// TIA Portal V17 export
// export: Created 2022-07-20T06:59:51.5033587Z, ExportSetting WithDefaults, DisplayName Totally Integrated Automation Portal, DisplayVersion V17, DisplayName TIA Portal Openness, DisplayVersion V17, DisplayName TIA Portal Version Control Interface, DisplayVersion V17, DisplayName SINAMICS Startdrive Advanced, DisplayVersion V17, DisplayName SINAMICS Startdrive G130, G150, S120, S150, SINAMICS MV, S210, DisplayVersion V17, DisplayName SINAMICS Startdrive G110M, G120, G120C, G120D, G120P, G115D, DisplayVersion V17, DisplayName STEP 7 Professional, DisplayVersion V17, DisplayName STEP 7 Safety, DisplayVersion V17, DisplayName WinCC Advanced, DisplayVersion V17
FUNCTION_BLOCK "FB10064_IperCleaningTrays"   // FB10064, LAD
{ S7_Optimized_Access := 'TRUE' }
VERSION : 0.1
// stored: AutoNumber false, IsIECCheckEnabled false, IsRetainMemResEnabled false, MemoryReserve 100, SetENOAutomatically false, UDAEnableTagReadback false
   VAR_INPUT
      Acknowledge : Bool;
      DriveInLexium : "TLexium_MDrv_Drv2Plc";
      RequestAcknowledge : Bool;
      CleaningTray_HomingSensor : Bool;
      CleaningTray_PurgeTrayPositionSensor_1 : Bool;
      CleaningTray_PurgeTrayPositionSensor_2 : Bool;
      PurgeTray1_HomingPositionSensor : Bool;
      PurgeTray2_HomingPositionSensor : Bool;
      PurgeTray1_PurgePositionSensor : Bool;
      PurgeTray2_PurgePositionSensor : Bool;
      Motor_HoldCurrent : SInt;
      Motor_RunCurrent : SInt;
      Motor_MmByMotorTurn : Real;
      Motor_HomingSpeedMmBySec : Real;
      Motor_SpeedMmBySec : Real;
      Motor_AccelerationMmBySec2 : DInt;
      Motor_DecelerationMmBySec2 : DInt;
      Motor_JogSpeedMmBySec : Real;
      Motor_RequestStop : Bool;
      CleaningTray_HomingPosition : Real;
      CleaningTray_CleaningPosition_1 : Real;
      CleaningTray_CleaningPosition_2 : Real;
      CleaningTray_WipingPosition_1 : Real;
      CleaningTray_WipingPosition_2 : Real;
      CleaningTray_RequestHoming : Bool;
      CleaningTray_RequestGoToOriginPosition : Bool;
      CleaningTray_RequestGoToCleaningPosition_1 : Bool;
      CleaningTray_RequestGoToCleaningPosition_2 : Bool;
      CleaningTray_RequestGoToWipingPosition_1 : Bool;
      CleaningTray_RequestGoToWipingPosition_2 : Bool;
      PurgeTray_RequestGotoHomingPosition : Bool;
      PurgeTray_RequestGoToPurgePosition : Bool;
   END_VAR
   VAR_OUTPUT
      CleaningTray_ActivePurgeTraySolenoidValveClutch_1 : Bool;
      CleaningTray_ActivePurgeTraySolenoidValveClutch_2 : Bool;
      CleaningTray_ActualPosition : Real;
      CleaningTray_HomingDone : Bool;
      CleaningTray_InOriginPosition : Bool;
      CleaningTray_InCleaningPosition_1 : Bool;
      CleaningTray_InCleaningPosition_2 : Bool;
      CleaningTray_InWipingPosition_1 : Bool;
      CleaningTray_InWipingPosition_2 : Bool;
      PurgeTray_HomingDone : Bool;
      PurgeTray_InHomingPosition : Bool;
      PurgeTray_InPurgePosition : Bool;
      CleaningTrayMotor_InError : Bool;
      CleaningTrayProcess_InError : Bool;
      CleaningTrayMotor_ErrorCode : Array[0..9] of UInt;
      Clutch_IsInPosition : Bool;
      Clutch_IsOutPosition : Bool;
   END_VAR
   VAR_IN_OUT
      DriveOutLexium : "TLexium_MDrv_Plc2Drv";
      Clutch_RequestIn : Bool;
      Clutch_RequestOut : Bool;
   END_VAR
   VAR
      Motor_Struct : Struct
         In : Struct
            UnitByTurn : LReal;
            HoldCurrent : SInt;
            RunCurrent : SInt;
            Speed_UnitBySec : Real;
            HomingSpeed_UnitBySec : Real;
            Acceleration_UnitBySec2 : Real;
            Deceleration_UnitBySec2 : Real;
            JogSpeed_MmBySec : Real;
            RequestHoming : Bool;
            RequestGoToPosition_1 : Bool;
            Position_1 : Real;
            RequestGoToPosition_2 : Bool;
            Position_2 : Real;
            RequestGoToPosition_3 : Bool;
            Position_3 : Real;
            RequestGoToPosition_4 : Bool;
            Position_4 : Real;
            RequestGoToPosition_5 : Bool;
            Position_5 : Real;
            RequestJogPositive : Bool;
            RequestJogNegative : Bool;
            RequestStop : Bool;
            Ack : Bool;
         END_STRUCT;
         Out : Struct
            ActualPosition : Real;
            HomingDone : Bool;
            IsInPosition_1 : Bool;
            IsInPosition_2 : Bool;
            IsInPosition_3 : Bool;
            IsInPosition_4 : Bool;
            IsInPosition_5 : Bool;
            InError : Bool;
            ErrorCode : Array[0..9] of UInt;
         END_STRUCT;
      END_STRUCT;
      SendNewRequestOk : Bool;
      MotorMovementManagementStateDiagram : Int;
      ClutchMovementManagementStateDiagram : Int;
      R_TRIG_CleaningTray_HomingSensor : R_TRIG;
      R_TRIG_CleaningTray_RequestHoming : R_TRIG;
      R_TRIG_CleaningTray_RequestGoToHomingPosition : R_TRIG;
      R_TRIG_CleaningTray_RequestGoToCleaningPosition_1 : R_TRIG;
      R_TRIG_CleaningTray_RequestGoToCleaningPosition_2 : R_TRIG;
      R_TRIG_CleaningTray_RequestGoToWipingPosition_1 : R_TRIG;
      R_TRIG_CleaningTray_RequestGoToWipingPosition_2 : R_TRIG;
      R_TRIG_PurgeTray_RequestGoToHomingPosition { S7_SetPoint := 'True'} : R_TRIG;
      R_TRIG_PurgeTray_RequestGoToPurgePosition : R_TRIG;
      R_TRIG_HomingDone { S7_SetPoint := 'True'} : R_TRIG;
      R_TRIG_Clutch_RequestIn { S7_SetPoint := 'True'} : R_TRIG;
      R_TRIG_Clutch_RequestOut { S7_SetPoint := 'True'} : R_TRIG;
      F_TRIG_CleaningTray_HomingSensor { S7_SetPoint := 'True'} : F_TRIG;
      F_TRIG_PurgeTray1_HomingPositionSensor : F_TRIG;
      F_TRIG_PurgeTray2_HomingPositionSensor : F_TRIG;
      F_TRIG_PurgeTray1_PurgePositionSensor : F_TRIG;
      F_TRIG_PurgeTray2_PurgePositionSensor : F_TRIG;
      F_TRIG_CleaningTray_PurgeTrayPositionSensor_1 : F_TRIG;
      F_TRIG_CleaningTray_PurgeTrayPositionSensor_2 : F_TRIG;
      TON_MovingTrayProcedureTimeout { S7_SetPoint := 'True'} : TON_TIME;
      TON_CleaningTrayMotor_SendNewRequest { S7_SetPoint := 'True'} : TON_TIME;
      TON_Clutch_ExhaustTime { S7_SetPoint := 'True'} : TON_TIME;
      "TON_Clutch_In/Out" { S7_SetPoint := 'True'} : TON_TIME;
      TON_NotHomingSensor { S7_SetPoint := 'True'} : TON_TIME;
      FB10234_LexiumMotor_Instance { S7_SetPoint := 'True'} : "FB10234_LexiumMotor";
   END_VAR
   VAR CONSTANT
      WAIT_FOR_MOTOR_MOVEMENT_REQUESTS : Int := 0;
      CLEANING_TRAY_HOMING_GET_OUT_THE_HOMING_SENSOR : Int := 10;
      CLEANING_TRAY_DO_HOMING : Int := 20;
      CLEANING_TRAY_GO_TO_HOMING_POSITION : Int := 30;
      CLEANING_TRAY_GO_TO_CLEANING_POSITION_1 : Int := 40;
      CLEANING_TRAY_GO_TO_WIPING_POSITION_1 : Int := 50;
      CLEANING_TRAY_GO_TO_CLEANING_POSITION_2 : Int := 60;
      CLEANING_TRAY_GO_TO_WIPING_POSITION_2 : Int := 70;
      PURGE_TRAY_HOMING_POSITION_INITIALIZE_MOTOR_POSITION : Int := 80;
      PURGE_TRAY_HOMING_POSITION_LOOK_FOR_PT_1 : Int := 90;
      PURGE_TRAY_HOMING_POSITION_BRING_BACK_PT_1 : Int := 100;
      PURGE_TRAY_HOMING_POSITION_LOOK_FOR_PT_2 : Int := 110;
      PURGE_TRAY_HOMING_POSITION_BRING_BACK_PT_2 : Int := 120;
      PURGE_TRAY_PURGE_POSITION_INITIALIZE_MOTOR_POSITION : Int := 130;
      PURGE_TRAY_PURGE_POSITION_LOOK_FOR_PT_2 : Int := 140;
      PURGE_TRAY_PURGE_POSITION_LOOK_FOR_PT_1 : Int := 150;
      PURGE_TRAY_PURGE_POSITION_BRING_PT_2 : Int := 160;
      PURGE_TRAY_PURGE_POSITION_BRING_PT_1 : Int := 170;
      MOTOR_MOVEMENT_REQUEST_DONE : Int := 180;
      "==========" : Bool;
      WAIT_FOR_CLUTCH_REQUEST : Int := 0;
      CLUTCH_OUT_EXHAUST_AIR : Int := 10;
      CLUTCH_OUT : Int := 20;
      CLUTCH_IN_EXHAUST_AIR : Int := 30;
      CLUTCH_IN : Int := 40;
      CLUTCH_REQUEST_DONE : Int := 50;
      "==========_1" : Bool;
   END_VAR
BEGIN

REGION Network 1 (SCL): First Scan
   IF "FirstScan" THEN
       #Motor_Struct.In.RequestHoming := FALSE;
       #Motor_Struct.In.RequestJogPositive := FALSE;
       #Motor_Struct.In.RequestJogNegative := FALSE;
       #Motor_Struct.In.RequestGoToPosition_1 := FALSE;
       #Motor_Struct.In.RequestGoToPosition_2 := FALSE;
       #Motor_Struct.In.RequestGoToPosition_3 := FALSE;
       #Motor_Struct.In.RequestGoToPosition_4 := FALSE;
       #Motor_Struct.In.RequestGoToPosition_5 := FALSE;
       #Motor_Struct.In.RequestStop := FALSE;
       #CleaningTray_HomingDone := FALSE;
       #CleaningTray_InOriginPosition := FALSE;
       #CleaningTray_InCleaningPosition_1 := FALSE;
       #CleaningTray_InCleaningPosition_2 := FALSE;
       #CleaningTray_InWipingPosition_1 := FALSE;
       #CleaningTray_InWipingPosition_2 := FALSE;
       #PurgeTray_InHomingPosition := FALSE;
       #PurgeTray_InPurgePosition := FALSE;
       #Clutch_RequestIn := FALSE;
       #Clutch_RequestOut := FALSE;
       #Clutch_IsInPosition := FALSE;
       #Clutch_IsOutPosition := FALSE;
       #SendNewRequestOk := FALSE;
       #MotorMovementManagementStateDiagram := #WAIT_FOR_MOTOR_MOVEMENT_REQUESTS;
   END_IF;
END_REGION

REGION Network 2 (SCL): Edge Signals & Timers
   REGION EDGE SIGNALS
       #R_TRIG_CleaningTray_HomingSensor(CLK := #CleaningTray_HomingSensor);
       #R_TRIG_CleaningTray_RequestHoming(CLK := #CleaningTray_RequestHoming);
       #R_TRIG_CleaningTray_RequestGoToHomingPosition(CLK := #CleaningTray_RequestGoToOriginPosition);
       #R_TRIG_CleaningTray_RequestGoToCleaningPosition_1(CLK := #CleaningTray_RequestGoToCleaningPosition_1);
       #R_TRIG_CleaningTray_RequestGoToCleaningPosition_2(CLK := #CleaningTray_RequestGoToCleaningPosition_2);
       #R_TRIG_CleaningTray_RequestGoToWipingPosition_1(CLK := #CleaningTray_RequestGoToWipingPosition_1);
       #R_TRIG_CleaningTray_RequestGoToWipingPosition_2(CLK := #CleaningTray_RequestGoToWipingPosition_2);
       #R_TRIG_PurgeTray_RequestGoToHomingPosition(CLK := #PurgeTray_RequestGotoHomingPosition);
       #R_TRIG_PurgeTray_RequestGoToPurgePosition(CLK := #PurgeTray_RequestGoToPurgePosition);
       #R_TRIG_HomingDone(CLK := #Motor_Struct.Out.HomingDone);
       #R_TRIG_Clutch_RequestIn(CLK := #Clutch_RequestIn);
       #R_TRIG_Clutch_RequestOut(CLK := #Clutch_RequestOut);

       #F_TRIG_CleaningTray_HomingSensor(CLK := #CleaningTray_HomingSensor);
       #F_TRIG_PurgeTray1_HomingPositionSensor(CLK := #PurgeTray1_HomingPositionSensor);
       #F_TRIG_PurgeTray2_HomingPositionSensor(CLK := #PurgeTray2_HomingPositionSensor);
       #F_TRIG_PurgeTray1_PurgePositionSensor(CLK := #PurgeTray1_PurgePositionSensor);
       #F_TRIG_PurgeTray2_PurgePositionSensor(CLK := #PurgeTray2_PurgePositionSensor);
       #F_TRIG_CleaningTray_PurgeTrayPositionSensor_1(CLK := #CleaningTray_PurgeTrayPositionSensor_1);
       #F_TRIG_CleaningTray_PurgeTrayPositionSensor_2(CLK := #CleaningTray_PurgeTrayPositionSensor_2);
   END_REGION

   REGION TIMERS
       #TON_CleaningTrayMotor_SendNewRequest(IN := #MotorMovementManagementStateDiagram = #CLEANING_TRAY_HOMING_GET_OUT_THE_HOMING_SENSOR OR
                                             #MotorMovementManagementStateDiagram = #CLEANING_TRAY_DO_HOMING OR
                                             #MotorMovementManagementStateDiagram = #CLEANING_TRAY_GO_TO_HOMING_POSITION OR
                                             #MotorMovementManagementStateDiagram = #CLEANING_TRAY_GO_TO_CLEANING_POSITION_1 OR
                                             #MotorMovementManagementStateDiagram = #CLEANING_TRAY_GO_TO_WIPING_POSITION_1 OR
                                             #MotorMovementManagementStateDiagram = #CLEANING_TRAY_GO_TO_CLEANING_POSITION_2 OR
                                             #MotorMovementManagementStateDiagram = #CLEANING_TRAY_GO_TO_WIPING_POSITION_2 OR
                                             #MotorMovementManagementStateDiagram = #PURGE_TRAY_HOMING_POSITION_INITIALIZE_MOTOR_POSITION OR
                                             #MotorMovementManagementStateDiagram = #PURGE_TRAY_HOMING_POSITION_LOOK_FOR_PT_1 OR
                                             #MotorMovementManagementStateDiagram = #PURGE_TRAY_HOMING_POSITION_BRING_BACK_PT_1 OR
                                             #MotorMovementManagementStateDiagram = #PURGE_TRAY_HOMING_POSITION_LOOK_FOR_PT_2 OR
                                             #MotorMovementManagementStateDiagram = #PURGE_TRAY_HOMING_POSITION_BRING_BACK_PT_2 OR
                                             #MotorMovementManagementStateDiagram = #PURGE_TRAY_PURGE_POSITION_INITIALIZE_MOTOR_POSITION OR
                                             #MotorMovementManagementStateDiagram = #PURGE_TRAY_PURGE_POSITION_LOOK_FOR_PT_2 OR
                                             #MotorMovementManagementStateDiagram = #PURGE_TRAY_PURGE_POSITION_LOOK_FOR_PT_1 OR
                                             #MotorMovementManagementStateDiagram = #PURGE_TRAY_PURGE_POSITION_BRING_PT_2 OR
                                             #MotorMovementManagementStateDiagram = #PURGE_TRAY_PURGE_POSITION_BRING_PT_1,
                                             PT := T#2s);
       #TON_Clutch_ExhaustTime(IN := #ClutchMovementManagementStateDiagram = #CLUTCH_OUT_EXHAUST_AIR OR
                               #ClutchMovementManagementStateDiagram = #CLUTCH_IN_EXHAUST_AIR,
                               PT := T#500ms);
       #"TON_Clutch_In/Out"(IN := #ClutchMovementManagementStateDiagram = #CLUTCH_IN OR
                            #ClutchMovementManagementStateDiagram = #CLUTCH_OUT,
                            PT := T#2s);
       #TON_NotHomingSensor(IN := NOT(#CleaningTray_HomingSensor),
                            PT := T#200ms);
       #TON_MovingTrayProcedureTimeout(IN := #MotorMovementManagementStateDiagram = #PURGE_TRAY_HOMING_POSITION_INITIALIZE_MOTOR_POSITION OR
                                       #MotorMovementManagementStateDiagram = #PURGE_TRAY_PURGE_POSITION_INITIALIZE_MOTOR_POSITION,
                                       PT := T#60s);
   END_REGION
END_REGION

REGION Network 3 (SCL): Cleaning Tray Commands Management
   //Motor Parameters Management
   #Motor_Struct.In.HoldCurrent := #Motor_HoldCurrent;
   #Motor_Struct.In.RunCurrent := #Motor_RunCurrent;
   #Motor_Struct.In.UnitByTurn := #Motor_MmByMotorTurn;
   #Motor_Struct.In.HomingSpeed_UnitBySec := #Motor_HomingSpeedMmBySec;
   #Motor_Struct.In.Speed_UnitBySec := #Motor_SpeedMmBySec;
   #Motor_Struct.In.Acceleration_UnitBySec2 := #Motor_AccelerationMmBySec2;
   #Motor_Struct.In.Deceleration_UnitBySec2 := #Motor_DecelerationMmBySec2;
   #Motor_Struct.In.JogSpeed_MmBySec := #Motor_JogSpeedMmBySec;

   //Motor Positions Management
   #Motor_Struct.In.Position_1 := #CleaningTray_HomingPosition;
   #Motor_Struct.In.Position_2 := #CleaningTray_CleaningPosition_1;
   #Motor_Struct.In.Position_3 := #CleaningTray_WipingPosition_1;
   #Motor_Struct.In.Position_4 := #CleaningTray_CleaningPosition_2;
   #Motor_Struct.In.Position_5 := #CleaningTray_WipingPosition_2;



   //Motor Requests Management
   #Motor_Struct.In.RequestStop := #Motor_RequestStop;
   #Motor_Struct.In.Ack := #RequestAcknowledge;

   //Motor Send New Request Management
   IF #TON_CleaningTrayMotor_SendNewRequest.Q THEN
       #SendNewRequestOk := TRUE;
   END_IF;
END_REGION

REGION Network 4: Cleaning Motor Tray Management
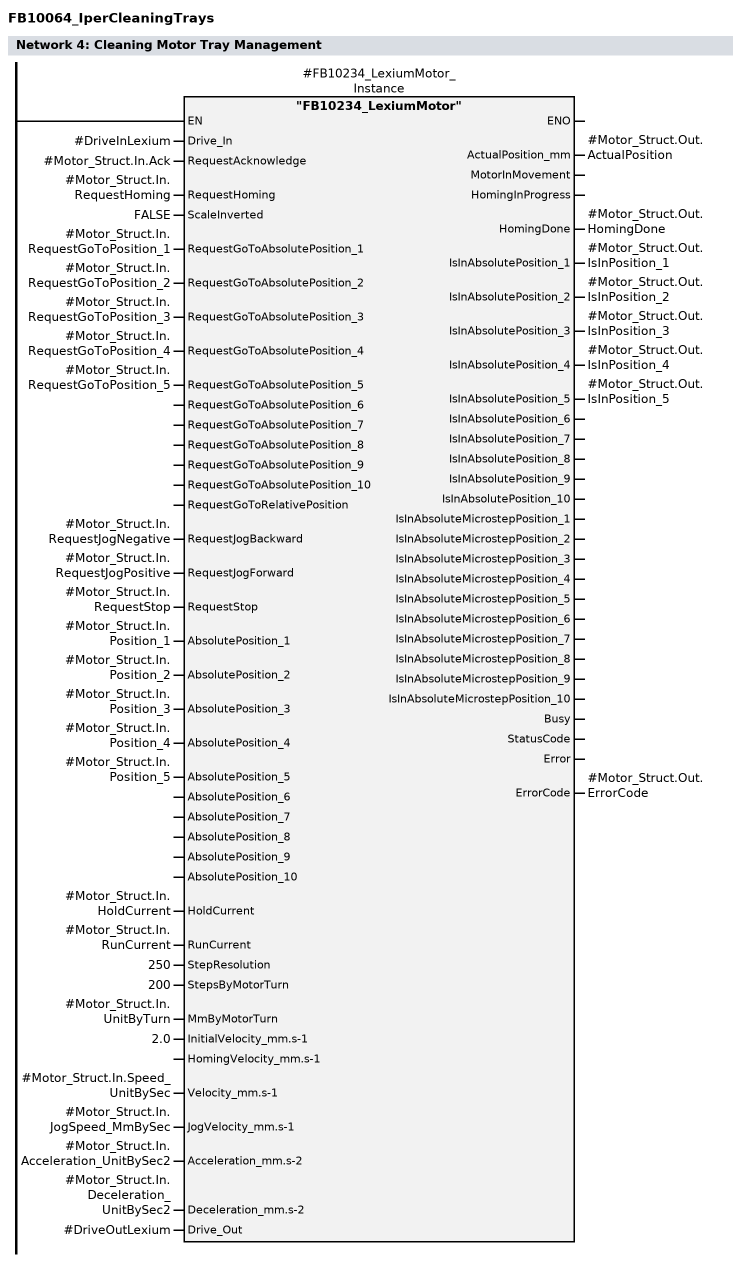
   RUNG wire#powerrail
      #FB10234_LexiumMotor_Instance(Drive_In := #DriveInLexium, RequestAcknowledge := #Motor_Struct.In.Ack, RequestHoming := #Motor_Struct.In.RequestHoming, ScaleInverted := FALSE, RequestGoToAbsolutePosition_1 := #Motor_Struct.In.RequestGoToPosition_1, RequestGoToAbsolutePosition_2 := #Motor_Struct.In.RequestGoToPosition_2, RequestGoToAbsolutePosition_3 := #Motor_Struct.In.RequestGoToPosition_3, RequestGoToAbsolutePosition_4 := #Motor_Struct.In.RequestGoToPosition_4, RequestGoToAbsolutePosition_5 := #Motor_Struct.In.RequestGoToPosition_5, RequestGoToAbsolutePosition_6 :=, RequestGoToAbsolutePosition_7 :=, RequestGoToAbsolutePosition_8 :=, RequestGoToAbsolutePosition_9 :=, RequestGoToAbsolutePosition_10 :=, RequestGoToRelativePosition :=, RequestJogBackward := #Motor_Struct.In.RequestJogNegative, RequestJogForward := #Motor_Struct.In.RequestJogPositive, RequestStop := #Motor_Struct.In.RequestStop, AbsolutePosition_1 := #Motor_Struct.In.Position_1, AbsolutePosition_2 := #Motor_Struct.In.Position_2, AbsolutePosition_3 := #Motor_Struct.In.Position_3, AbsolutePosition_4 := #Motor_Struct.In.Position_4, AbsolutePosition_5 := #Motor_Struct.In.Position_5, AbsolutePosition_6 :=, AbsolutePosition_7 :=, AbsolutePosition_8 :=, AbsolutePosition_9 :=, AbsolutePosition_10 :=, HoldCurrent := #Motor_Struct.In.HoldCurrent, RunCurrent := #Motor_Struct.In.RunCurrent, StepResolution := 250, StepsByMotorTurn := 200, MmByMotorTurn := #Motor_Struct.In.UnitByTurn, "InitialVelocity_mm.s-1" := 2.0, "HomingVelocity_mm.s-1" :=, "Velocity_mm.s-1" := #Motor_Struct.In.Speed_UnitBySec, "JogVelocity_mm.s-1" := #Motor_Struct.In.JogSpeed_MmBySec, "Acceleration_mm.s-2" := #Motor_Struct.In.Acceleration_UnitBySec2, "Deceleration_mm.s-2" := #Motor_Struct.In.Deceleration_UnitBySec2, Drive_Out := #DriveOutLexium, ActualPosition_mm => #Motor_Struct.Out.ActualPosition, MotorInMovement =>, HomingInProgress =>, HomingDone => #Motor_Struct.Out.HomingDone, IsInAbsolutePosition_1 => #Motor_Struct.Out.IsInPosition_1, IsInAbsolutePosition_2 => #Motor_Struct.Out.IsInPosition_2, IsInAbsolutePosition_3 => #Motor_Struct.Out.IsInPosition_3, IsInAbsolutePosition_4 => #Motor_Struct.Out.IsInPosition_4, IsInAbsolutePosition_5 => #Motor_Struct.Out.IsInPosition_5, IsInAbsolutePosition_6 =>, IsInAbsolutePosition_7 =>, IsInAbsolutePosition_8 =>, IsInAbsolutePosition_9 =>, IsInAbsolutePosition_10 =>, IsInAbsoluteMicrostepPosition_1 =>, IsInAbsoluteMicrostepPosition_2 =>, IsInAbsoluteMicrostepPosition_3 =>, IsInAbsoluteMicrostepPosition_4 =>, IsInAbsoluteMicrostepPosition_5 =>, IsInAbsoluteMicrostepPosition_6 =>, IsInAbsoluteMicrostepPosition_7 =>, IsInAbsoluteMicrostepPosition_8 =>, IsInAbsoluteMicrostepPosition_9 =>, IsInAbsoluteMicrostepPosition_10 =>, Busy =>, StatusCode =>, Error =>, ErrorCode => #Motor_Struct.Out.ErrorCode)
   END_RUNG
   // the same network as SCL:
   #FB10234_LexiumMotor_Instance(Drive_In := #DriveInLexium,   // "FB10234_LexiumMotor"
                           RequestAcknowledge := #Motor_Struct.In.Ack,
                           RequestHoming := #Motor_Struct.In.RequestHoming,
                           ScaleInverted := FALSE,
                           RequestGoToAbsolutePosition_1 := #Motor_Struct.In.RequestGoToPosition_1,
                           RequestGoToAbsolutePosition_2 := #Motor_Struct.In.RequestGoToPosition_2,
                           RequestGoToAbsolutePosition_3 := #Motor_Struct.In.RequestGoToPosition_3,
                           RequestGoToAbsolutePosition_4 := #Motor_Struct.In.RequestGoToPosition_4,
                           RequestGoToAbsolutePosition_5 := #Motor_Struct.In.RequestGoToPosition_5,
                           RequestJogBackward := #Motor_Struct.In.RequestJogNegative,
                           RequestJogForward := #Motor_Struct.In.RequestJogPositive,
                           RequestStop := #Motor_Struct.In.RequestStop,
                           AbsolutePosition_1 := #Motor_Struct.In.Position_1,
                           AbsolutePosition_2 := #Motor_Struct.In.Position_2,
                           AbsolutePosition_3 := #Motor_Struct.In.Position_3,
                           AbsolutePosition_4 := #Motor_Struct.In.Position_4,
                           AbsolutePosition_5 := #Motor_Struct.In.Position_5,
                           HoldCurrent := #Motor_Struct.In.HoldCurrent,
                           RunCurrent := #Motor_Struct.In.RunCurrent,
                           StepResolution := 250,
                           StepsByMotorTurn := 200,
                           MmByMotorTurn := #Motor_Struct.In.UnitByTurn,
                           "InitialVelocity_mm.s-1" := 2.0,
                           "Velocity_mm.s-1" := #Motor_Struct.In.Speed_UnitBySec,
                           "JogVelocity_mm.s-1" := #Motor_Struct.In.JogSpeed_MmBySec,
                           "Acceleration_mm.s-2" := #Motor_Struct.In.Acceleration_UnitBySec2,
                           "Deceleration_mm.s-2" := #Motor_Struct.In.Deceleration_UnitBySec2,
                           Drive_Out := #DriveOutLexium,
                           ActualPosition_mm => #Motor_Struct.Out.ActualPosition,
                           HomingDone => #Motor_Struct.Out.HomingDone,
                           IsInAbsolutePosition_1 => #Motor_Struct.Out.IsInPosition_1,
                           IsInAbsolutePosition_2 => #Motor_Struct.Out.IsInPosition_2,
                           IsInAbsolutePosition_3 => #Motor_Struct.Out.IsInPosition_3,
                           IsInAbsolutePosition_4 => #Motor_Struct.Out.IsInPosition_4,
                           IsInAbsolutePosition_5 => #Motor_Struct.Out.IsInPosition_5,
                           ErrorCode => #Motor_Struct.Out.ErrorCode);
END_REGION

REGION Network 5 (SCL): Motor Movement Management
   IF #Motor_RequestStop THEN
       #MotorMovementManagementStateDiagram := #WAIT_FOR_MOTOR_MOVEMENT_REQUESTS;
       #Motor_Struct.In.RequestHoming := FALSE;
       #Motor_Struct.In.RequestJogPositive := FALSE;
       #Motor_Struct.In.RequestJogNegative := FALSE;
       #Motor_Struct.In.RequestGoToPosition_1 := FALSE;
       #Motor_Struct.In.RequestGoToPosition_2 := FALSE;
       #Motor_Struct.In.RequestGoToPosition_3 := FALSE;
       #Motor_Struct.In.RequestGoToPosition_4 := FALSE;
       #Motor_Struct.In.RequestGoToPosition_5 := FALSE;
   END_IF;

   CASE #MotorMovementManagementStateDiagram OF
       #WAIT_FOR_MOTOR_MOVEMENT_REQUESTS:
           IF #R_TRIG_CleaningTray_RequestHoming.Q THEN
               #CleaningTray_HomingDone := FALSE;
               #MotorMovementManagementStateDiagram := #CLEANING_TRAY_DO_HOMING;
           ELSIF #R_TRIG_CleaningTray_RequestGoToHomingPosition.Q THEN
               #CleaningTray_InOriginPosition := FALSE;
               #MotorMovementManagementStateDiagram := #CLEANING_TRAY_GO_TO_HOMING_POSITION;
           ELSIF #R_TRIG_CleaningTray_RequestGoToCleaningPosition_1.Q THEN
               #CleaningTray_InCleaningPosition_1 := FALSE;
               #MotorMovementManagementStateDiagram := #CLEANING_TRAY_GO_TO_CLEANING_POSITION_1;
           ELSIF #R_TRIG_CleaningTray_RequestGoToWipingPosition_1.Q THEN
               #CleaningTray_InWipingPosition_1 := FALSE;
               #MotorMovementManagementStateDiagram := #CLEANING_TRAY_GO_TO_WIPING_POSITION_1;
           ELSIF #R_TRIG_CleaningTray_RequestGoToCleaningPosition_2.Q THEN
               #CleaningTray_InCleaningPosition_2 := FALSE;
               #MotorMovementManagementStateDiagram := #CLEANING_TRAY_GO_TO_CLEANING_POSITION_2;
           ELSIF #R_TRIG_CleaningTray_RequestGoToWipingPosition_2.Q THEN
               #CleaningTray_InWipingPosition_2 := FALSE;
               #MotorMovementManagementStateDiagram := #CLEANING_TRAY_GO_TO_WIPING_POSITION_2;
           ELSIF #R_TRIG_PurgeTray_RequestGoToHomingPosition.Q THEN
               #PurgeTray_InHomingPosition := FALSE;
               #MotorMovementManagementStateDiagram := #PURGE_TRAY_HOMING_POSITION_INITIALIZE_MOTOR_POSITION;
           ELSIF #R_TRIG_PurgeTray_RequestGoToPurgePosition.Q THEN
               #PurgeTray_InPurgePosition := FALSE;
               #MotorMovementManagementStateDiagram := #PURGE_TRAY_PURGE_POSITION_INITIALIZE_MOTOR_POSITION;
           END_IF;
       #CLEANING_TRAY_HOMING_GET_OUT_THE_HOMING_SENSOR:
           IF #Clutch_IsInPosition AND #SendNewRequestOk THEN
               #Clutch_RequestIn := FALSE;
               #Motor_Struct.In.RequestJogPositive := TRUE;
               IF #F_TRIG_CleaningTray_HomingSensor.Q THEN
                   #Motor_Struct.In.RequestJogPositive := FALSE;
                   #SendNewRequestOk := FALSE;
                   RESET_TIMER(#TON_CleaningTrayMotor_SendNewRequest);
                   #MotorMovementManagementStateDiagram := #CLEANING_TRAY_DO_HOMING;
               END_IF;
           ELSE
               #Clutch_RequestIn := TRUE;
           END_IF;
       #CLEANING_TRAY_DO_HOMING:
           IF #Clutch_IsInPosition AND #SendNewRequestOk THEN
               #Clutch_RequestIn := FALSE;
               #Motor_Struct.In.RequestHoming := TRUE;
               IF #R_TRIG_HomingDone.Q THEN
                   #Motor_Struct.In.RequestHoming := FALSE;
                   #CleaningTray_HomingDone := TRUE;
                   #SendNewRequestOk := FALSE;
                   RESET_TIMER(#TON_CleaningTrayMotor_SendNewRequest);
                   #MotorMovementManagementStateDiagram := #MOTOR_MOVEMENT_REQUEST_DONE;
               END_IF;
           ELSE
               #Clutch_RequestIn := TRUE;
           END_IF;
       #CLEANING_TRAY_GO_TO_HOMING_POSITION:
           IF #Clutch_IsInPosition AND #SendNewRequestOk THEN
               #Clutch_RequestIn := FALSE;
               #Motor_Struct.In.RequestGoToPosition_1 := TRUE;
               IF #Motor_Struct.Out.IsInPosition_1 THEN
                   #Motor_Struct.In.RequestGoToPosition_1 := FALSE;
                   #SendNewRequestOk := FALSE;
                   RESET_TIMER(#TON_CleaningTrayMotor_SendNewRequest);
                   #MotorMovementManagementStateDiagram := #MOTOR_MOVEMENT_REQUEST_DONE;
               END_IF;
           ELSE
               #Clutch_RequestIn := TRUE;
           END_IF;
       #CLEANING_TRAY_GO_TO_CLEANING_POSITION_1:
           IF #Clutch_IsInPosition AND #SendNewRequestOk THEN
               #Clutch_RequestIn := FALSE;
               #Motor_Struct.In.RequestGoToPosition_2 := TRUE;
               IF #Motor_Struct.Out.IsInPosition_2 THEN
                   #Motor_Struct.In.RequestGoToPosition_2 := FALSE;
                   #SendNewRequestOk := FALSE;
                   RESET_TIMER(#TON_CleaningTrayMotor_SendNewRequest);
                   #MotorMovementManagementStateDiagram := #MOTOR_MOVEMENT_REQUEST_DONE;
               END_IF;
           ELSE
               #Clutch_RequestIn := TRUE;
           END_IF;
       #CLEANING_TRAY_GO_TO_WIPING_POSITION_1:
           IF #Clutch_IsInPosition AND #SendNewRequestOk THEN
               #Clutch_RequestIn := FALSE;
               #Motor_Struct.In.RequestGoToPosition_3 := TRUE;
               IF #Motor_Struct.Out.IsInPosition_3 THEN
                   #Motor_Struct.In.RequestGoToPosition_3 := FALSE;
                   #SendNewRequestOk := FALSE;
                   RESET_TIMER(#TON_CleaningTrayMotor_SendNewRequest);
                   #MotorMovementManagementStateDiagram := #MOTOR_MOVEMENT_REQUEST_DONE;
               END_IF;
           ELSE
               #Clutch_RequestIn := TRUE;
           END_IF;
       #CLEANING_TRAY_GO_TO_CLEANING_POSITION_2:
           IF #Clutch_IsInPosition AND #SendNewRequestOk THEN
               #Clutch_RequestIn := FALSE;
               #Motor_Struct.In.RequestGoToPosition_4 := TRUE;
               IF #Motor_Struct.Out.IsInPosition_4 THEN
                   #Motor_Struct.In.RequestGoToPosition_4 := FALSE;
                   #SendNewRequestOk := FALSE;
                   RESET_TIMER(#TON_CleaningTrayMotor_SendNewRequest);
                   #MotorMovementManagementStateDiagram := #MOTOR_MOVEMENT_REQUEST_DONE;
               END_IF;
           ELSE
               #Clutch_RequestIn := TRUE;
           END_IF;
       #CLEANING_TRAY_GO_TO_WIPING_POSITION_2:
           #Motor_Struct.In.RequestGoToPosition_5 := TRUE;
           IF #Clutch_IsInPosition AND #SendNewRequestOk THEN
               #Clutch_RequestIn := FALSE;
               IF #Motor_Struct.Out.IsInPosition_5 THEN
                   #Motor_Struct.In.RequestGoToPosition_5 := FALSE;
                   #SendNewRequestOk := FALSE;
                   RESET_TIMER(#TON_CleaningTrayMotor_SendNewRequest);
                   #MotorMovementManagementStateDiagram := #MOTOR_MOVEMENT_REQUEST_DONE;
               END_IF;
           ELSE
               #Clutch_RequestIn := TRUE;
           END_IF;
       #PURGE_TRAY_HOMING_POSITION_INITIALIZE_MOTOR_POSITION:
           IF #Clutch_IsInPosition AND #SendNewRequestOk THEN
               #Clutch_RequestIn := FALSE;
               IF NOT (#PurgeTray1_HomingPositionSensor) AND NOT (#PurgeTray2_HomingPositionSensor) THEN // AND #CleaningTray_HomingSensor THEN //80.0 mm Distance Between Cleaning Tray Purge Tray 1 Sensor In Homing Position And Cleaning Tray Homing Sensor
                   #Motor_Struct.In.RequestJogNegative := FALSE;
                   #SendNewRequestOk := FALSE;
                   RESET_TIMER(#TON_CleaningTrayMotor_SendNewRequest);
                   #MotorMovementManagementStateDiagram := #CLEANING_TRAY_GO_TO_HOMING_POSITION;
               ELSIF #PurgeTray1_HomingPositionSensor AND #PurgeTray2_HomingPositionSensor AND #CleaningTray_HomingSensor THEN
                   #Motor_Struct.In.RequestJogNegative := FALSE;
                   #SendNewRequestOk := FALSE;
                   RESET_TIMER(#TON_CleaningTrayMotor_SendNewRequest);
                   #MotorMovementManagementStateDiagram := #PURGE_TRAY_HOMING_POSITION_LOOK_FOR_PT_1;
               ELSIF #PurgeTray1_HomingPositionSensor AND #F_TRIG_CleaningTray_PurgeTrayPositionSensor_1.Q THEN
                   #Motor_Struct.In.RequestJogNegative := FALSE;
                   #SendNewRequestOk := FALSE;
                   RESET_TIMER(#TON_CleaningTrayMotor_SendNewRequest);
                   #MotorMovementManagementStateDiagram := #PURGE_TRAY_HOMING_POSITION_BRING_BACK_PT_1;
               ELSIF NOT (#PurgeTray1_HomingPositionSensor) AND #PurgeTray2_HomingPositionSensor AND #CleaningTray_HomingSensor THEN
                   #Motor_Struct.In.RequestJogNegative := FALSE;
                   #SendNewRequestOk := FALSE;
                   RESET_TIMER(#TON_CleaningTrayMotor_SendNewRequest);
                   #MotorMovementManagementStateDiagram := #PURGE_TRAY_HOMING_POSITION_LOOK_FOR_PT_2;
               ELSIF NOT (#PurgeTray1_HomingPositionSensor) AND #PurgeTray2_HomingPositionSensor AND #F_TRIG_CleaningTray_PurgeTrayPositionSensor_2.Q THEN
                   #Motor_Struct.In.RequestJogNegative := FALSE;
                   #SendNewRequestOk := FALSE;
                   RESET_TIMER(#TON_CleaningTrayMotor_SendNewRequest);
                   #MotorMovementManagementStateDiagram := #PURGE_TRAY_HOMING_POSITION_BRING_BACK_PT_2;
               ELSIF NOT (#CleaningTray_HomingSensor) OR NOT(#Motor_Struct.Out.ActualPosition <= 5.0) THEN
                   #Motor_Struct.In.RequestJogNegative := TRUE;
               END_IF;
           ELSE
               #Clutch_RequestIn := TRUE;
           END_IF;
       #PURGE_TRAY_HOMING_POSITION_LOOK_FOR_PT_1:
           IF #Clutch_IsInPosition AND #SendNewRequestOk THEN
               #Clutch_RequestIn := FALSE;
               #Motor_Struct.In.RequestJogPositive := TRUE;
               IF #F_TRIG_CleaningTray_PurgeTrayPositionSensor_1.Q THEN
                   #Motor_Struct.In.RequestJogPositive := FALSE;
                   #SendNewRequestOk := FALSE;
                   RESET_TIMER(#TON_CleaningTrayMotor_SendNewRequest);
                   #MotorMovementManagementStateDiagram := #PURGE_TRAY_HOMING_POSITION_BRING_BACK_PT_1;
               END_IF;
           ELSE
               #Clutch_RequestIn := TRUE;
           END_IF;
       #PURGE_TRAY_HOMING_POSITION_BRING_BACK_PT_1:
           IF #Clutch_IsOutPosition AND #SendNewRequestOk THEN
               #Clutch_RequestOut := FALSE;
               #Motor_Struct.In.RequestJogNegative := TRUE;
               IF #F_TRIG_PurgeTray1_HomingPositionSensor.Q THEN
                   #Motor_Struct.In.RequestJogNegative := FALSE;
                   #SendNewRequestOk := FALSE;
                   RESET_TIMER(#TON_CleaningTrayMotor_SendNewRequest);
                   #MotorMovementManagementStateDiagram := #PURGE_TRAY_HOMING_POSITION_LOOK_FOR_PT_2;
               END_IF;
           ELSE
               #Clutch_RequestOut := TRUE;
           END_IF;
       #PURGE_TRAY_HOMING_POSITION_LOOK_FOR_PT_2:
           IF #Clutch_IsInPosition AND #SendNewRequestOk THEN
               #Clutch_RequestIn := FALSE;
               #Motor_Struct.In.RequestJogPositive := TRUE;
               IF #F_TRIG_CleaningTray_PurgeTrayPositionSensor_2.Q THEN
                   #Motor_Struct.In.RequestJogPositive := FALSE;
                   #SendNewRequestOk := FALSE;
                   RESET_TIMER(#TON_CleaningTrayMotor_SendNewRequest);
                   #MotorMovementManagementStateDiagram := #PURGE_TRAY_HOMING_POSITION_BRING_BACK_PT_2;
               END_IF;
           ELSE
               #Clutch_RequestIn := TRUE;
           END_IF;
       #PURGE_TRAY_HOMING_POSITION_BRING_BACK_PT_2:
           IF #Clutch_IsOutPosition AND #SendNewRequestOk THEN
               #Clutch_RequestOut := FALSE;
               #Motor_Struct.In.RequestJogNegative := TRUE;
               IF #F_TRIG_PurgeTray2_HomingPositionSensor.Q THEN
                   #Motor_Struct.In.RequestJogNegative := FALSE;
                   #SendNewRequestOk := FALSE;
                   RESET_TIMER(#TON_CleaningTrayMotor_SendNewRequest);
                   #MotorMovementManagementStateDiagram := #CLEANING_TRAY_GO_TO_HOMING_POSITION;
               END_IF;
           ELSE
               #Clutch_RequestOut := TRUE;
           END_IF;
       #PURGE_TRAY_PURGE_POSITION_INITIALIZE_MOTOR_POSITION:
           IF #Clutch_IsInPosition THEN
               #Clutch_RequestIn := FALSE;
               IF NOT (#PurgeTray1_PurgePositionSensor) AND NOT (#PurgeTray2_PurgePositionSensor) THEN //AND #CleaningTray_HomingSensor THEN
                   #Motor_Struct.In.RequestJogNegative := FALSE;
                   #SendNewRequestOk := FALSE;
                   RESET_TIMER(#TON_CleaningTrayMotor_SendNewRequest);
                   #MotorMovementManagementStateDiagram := #CLEANING_TRAY_GO_TO_HOMING_POSITION;
               ELSIF #PurgeTray1_PurgePositionSensor AND #PurgeTray2_PurgePositionSensor AND #CleaningTray_HomingSensor THEN
                   #Motor_Struct.In.RequestJogNegative := FALSE;
                   #SendNewRequestOk := FALSE;
                   RESET_TIMER(#TON_CleaningTrayMotor_SendNewRequest);
                   #MotorMovementManagementStateDiagram := #PURGE_TRAY_PURGE_POSITION_LOOK_FOR_PT_2;
               ELSIF #PurgeTray2_PurgePositionSensor AND #F_TRIG_CleaningTray_PurgeTrayPositionSensor_2.Q THEN
                   #Motor_Struct.In.RequestJogNegative := FALSE;
                   #SendNewRequestOk := FALSE;
                   RESET_TIMER(#TON_CleaningTrayMotor_SendNewRequest);
                   #MotorMovementManagementStateDiagram := #PURGE_TRAY_PURGE_POSITION_BRING_PT_2;
               ELSIF #PurgeTray1_PurgePositionSensor AND NOT (#PurgeTray2_PurgePositionSensor) AND (#CleaningTray_HomingSensor OR #CleaningTray_InOriginPosition) THEN
                   #Motor_Struct.In.RequestJogNegative := FALSE;
                   #SendNewRequestOk := FALSE;
                   RESET_TIMER(#TON_CleaningTrayMotor_SendNewRequest);
                   #MotorMovementManagementStateDiagram := #PURGE_TRAY_PURGE_POSITION_LOOK_FOR_PT_1;
               ELSIF #PurgeTray1_PurgePositionSensor AND NOT (#PurgeTray2_PurgePositionSensor) AND #F_TRIG_CleaningTray_PurgeTrayPositionSensor_1.Q THEN
                   #Motor_Struct.In.RequestJogNegative := FALSE;
                   #SendNewRequestOk := FALSE;
                   RESET_TIMER(#TON_CleaningTrayMotor_SendNewRequest);
                   #MotorMovementManagementStateDiagram := #PURGE_TRAY_PURGE_POSITION_BRING_PT_2;
               ELSIF NOT (#CleaningTray_HomingSensor) OR NOT (#CleaningTray_InOriginPosition) THEN
                   #Motor_Struct.In.RequestJogNegative := TRUE;
               END_IF;
           ELSE
               #Clutch_RequestIn := TRUE;
           END_IF;
       #PURGE_TRAY_PURGE_POSITION_LOOK_FOR_PT_2:
           IF #Clutch_IsInPosition AND #SendNewRequestOk THEN
               #Clutch_RequestIn := FALSE;
               #Motor_Struct.In.RequestJogPositive := TRUE;
               IF #F_TRIG_CleaningTray_PurgeTrayPositionSensor_2.Q THEN
                   #Motor_Struct.In.RequestJogPositive := FALSE;
                   #SendNewRequestOk := FALSE;
                   RESET_TIMER(#TON_CleaningTrayMotor_SendNewRequest);
                   #MotorMovementManagementStateDiagram := #PURGE_TRAY_PURGE_POSITION_BRING_PT_2;
               END_IF;
           ELSE
               #Clutch_RequestIn := TRUE;
           END_IF;
       #PURGE_TRAY_PURGE_POSITION_BRING_PT_2:
           IF #Clutch_IsOutPosition AND #SendNewRequestOk THEN
               #Clutch_RequestOut := FALSE;
               #Motor_Struct.In.RequestJogPositive := TRUE;
               IF #F_TRIG_PurgeTray2_PurgePositionSensor.Q THEN
                   #Motor_Struct.In.RequestJogPositive := FALSE;
                   #SendNewRequestOk := FALSE;
                   RESET_TIMER(#TON_CleaningTrayMotor_SendNewRequest);
                   #MotorMovementManagementStateDiagram := #PURGE_TRAY_PURGE_POSITION_LOOK_FOR_PT_1;
               END_IF;
           ELSE
               #Clutch_RequestOut := TRUE;
           END_IF;
       #PURGE_TRAY_PURGE_POSITION_LOOK_FOR_PT_1:
           IF #Clutch_IsInPosition AND #SendNewRequestOk THEN
               #Clutch_RequestIn := FALSE;
               #Motor_Struct.In.RequestJogNegative := TRUE;
               IF #F_TRIG_CleaningTray_PurgeTrayPositionSensor_1.Q THEN
                   #Motor_Struct.In.RequestJogNegative := FALSE;
                   #SendNewRequestOk := FALSE;
                   RESET_TIMER(#TON_CleaningTrayMotor_SendNewRequest);
                   #MotorMovementManagementStateDiagram := #PURGE_TRAY_PURGE_POSITION_BRING_PT_1;
               END_IF;
           ELSE
               #Clutch_RequestIn := TRUE;
           END_IF;
       #PURGE_TRAY_PURGE_POSITION_BRING_PT_1:
           IF #Clutch_IsOutPosition AND #SendNewRequestOk THEN
               #Clutch_RequestOut := FALSE;
               #Motor_Struct.In.RequestJogPositive := TRUE;
               IF #F_TRIG_PurgeTray1_PurgePositionSensor.Q THEN
                   #Motor_Struct.In.RequestJogPositive := FALSE;
                   #SendNewRequestOk := FALSE;
                   RESET_TIMER(#TON_CleaningTrayMotor_SendNewRequest);
                   #MotorMovementManagementStateDiagram := #CLEANING_TRAY_GO_TO_HOMING_POSITION;
               END_IF;
           ELSE
               #Clutch_RequestOut := TRUE;
           END_IF;
       #MOTOR_MOVEMENT_REQUEST_DONE:
           #MotorMovementManagementStateDiagram := #WAIT_FOR_MOTOR_MOVEMENT_REQUESTS;
   END_CASE;
END_REGION

REGION Network 6 (SCL): Clutch Movement Management
   CASE #ClutchMovementManagementStateDiagram OF
       #WAIT_FOR_CLUTCH_REQUEST:
           IF #R_TRIG_Clutch_RequestIn.Q THEN
               #Clutch_IsInPosition := FALSE;
               #Clutch_IsOutPosition := FALSE;
               #ClutchMovementManagementStateDiagram := #CLUTCH_IN_EXHAUST_AIR;
           ELSIF #R_TRIG_Clutch_RequestOut.Q THEN
               #Clutch_IsInPosition := FALSE;
               #Clutch_IsOutPosition := FALSE;
               #ClutchMovementManagementStateDiagram := #CLUTCH_OUT_EXHAUST_AIR;
           END_IF;
       #CLUTCH_OUT_EXHAUST_AIR:
           #CleaningTray_ActivePurgeTraySolenoidValveClutch_1 := TRUE;
           #CleaningTray_ActivePurgeTraySolenoidValveClutch_2 := FALSE;
           IF #TON_Clutch_ExhaustTime.Q THEN
               #ClutchMovementManagementStateDiagram := #CLUTCH_OUT;
           END_IF;
       #CLUTCH_OUT:
           #CleaningTray_ActivePurgeTraySolenoidValveClutch_1 := TRUE;
           #CleaningTray_ActivePurgeTraySolenoidValveClutch_2 := TRUE;
           IF #CleaningTray_ActivePurgeTraySolenoidValveClutch_1 AND #CleaningTray_ActivePurgeTraySolenoidValveClutch_2 AND #"TON_Clutch_In/Out".Q THEN
               #Clutch_IsOutPosition := TRUE;
               #ClutchMovementManagementStateDiagram := #CLUTCH_REQUEST_DONE;
           END_IF;
       #CLUTCH_IN_EXHAUST_AIR:
           #CleaningTray_ActivePurgeTraySolenoidValveClutch_1 := FALSE;
           #CleaningTray_ActivePurgeTraySolenoidValveClutch_2 := TRUE;
           IF #TON_Clutch_ExhaustTime.Q THEN
               #ClutchMovementManagementStateDiagram := #CLUTCH_IN;
           END_IF;
       #CLUTCH_IN:
           #CleaningTray_ActivePurgeTraySolenoidValveClutch_1 := FALSE;
           #CleaningTray_ActivePurgeTraySolenoidValveClutch_2 := FALSE;
           IF NOT (#CleaningTray_ActivePurgeTraySolenoidValveClutch_1) AND NOT (#CleaningTray_ActivePurgeTraySolenoidValveClutch_2) AND #"TON_Clutch_In/Out".Q THEN
               #Clutch_IsInPosition := TRUE;
               #ClutchMovementManagementStateDiagram := #CLUTCH_REQUEST_DONE;
           END_IF;
       #CLUTCH_REQUEST_DONE:
           #ClutchMovementManagementStateDiagram := #WAIT_FOR_CLUTCH_REQUEST;
   END_CASE;
END_REGION

REGION Network 7 (SCL): Motor Error Management
   IF #Motor_Struct.Out.InError THEN
       #MotorMovementManagementStateDiagram := #WAIT_FOR_MOTOR_MOVEMENT_REQUESTS;
       #Motor_Struct.In.Ack := #RequestAcknowledge;
       #Motor_Struct.In.RequestHoming := FALSE;
       #Motor_Struct.In.RequestJogPositive := FALSE;
       #Motor_Struct.In.RequestJogNegative := FALSE;
       #Motor_Struct.In.RequestGoToPosition_1 := FALSE;
       #Motor_Struct.In.RequestGoToPosition_2 := FALSE;
       #Motor_Struct.In.RequestGoToPosition_3 := FALSE;
       #Motor_Struct.In.RequestGoToPosition_4 := FALSE;
       #Motor_Struct.In.RequestGoToPosition_5 := FALSE;
       #SendNewRequestOk := FALSE;
   END_IF;
END_REGION

REGION Network 8 (SCL): Trays States Management
   //Motor Position States Management
   #CleaningTray_ActualPosition := #Motor_Struct.Out.ActualPosition;
   IF #CleaningTray_HomingSensor THEN
       #CleaningTray_InOriginPosition := TRUE;
   ELSIF #TON_NotHomingSensor.Q THEN
       #CleaningTray_InOriginPosition := FALSE;
   END_IF;
   #CleaningTray_InCleaningPosition_1 := #Motor_Struct.Out.IsInPosition_2;
   #CleaningTray_InWipingPosition_1 := #Motor_Struct.Out.IsInPosition_3;
   #CleaningTray_InCleaningPosition_2 := #Motor_Struct.Out.IsInPosition_4;
   #CleaningTray_InWipingPosition_2 := #Motor_Struct.Out.IsInPosition_5;

   //Purge Trays States Management
   #PurgeTray_InPurgePosition := NOT (#PurgeTray1_PurgePositionSensor) AND NOT (#PurgeTray2_PurgePositionSensor);
   #PurgeTray_InHomingPosition := NOT (#PurgeTray1_HomingPositionSensor) AND NOT (#PurgeTray2_HomingPositionSensor);
   //Motor Error States Management
   #CleaningTrayMotor_InError := #Motor_Struct.Out.InError;
   #CleaningTrayMotor_ErrorCode := #Motor_Struct.Out.ErrorCode;

   //Cleaning Tray Process In Error
   IF #TON_MovingTrayProcedureTimeout.Q THEN
       #CleaningTrayProcess_InError := TRUE;
   ELSIF #Acknowledge THEN
       #CleaningTrayProcess_InError := FALSE;
   END_IF;
END_REGION
END_FUNCTION_BLOCK
